TYPE IntSintBoolUnion :
UNION
	ValInt	:INT;
	ValSint :ARRAY[1..2] OF SINT;
	ValBool	:ARRAY[1..2] OF BitStructure;
END_UNION
END_TYPE

(* stored: Version 1.1.0.1, ProductVersion 3.1.4024.11
   DUT IntSintBoolUnion: Id {f56eed9b-d817-46fd-8e6b-9768f1393b44} *)
